(* IEC 61131-3 sources: programs/VI-54/VI-54_20171205/VI-54_20171205/Stations/Screen/LseClass170718/Class/AccessControlCreateAdmin, 1 file *)

(* ---- AccessControlCreateAdmin.st ---- *)
(*!
<Class
	Name               = "AccessControlCreateAdmin"
	Revision           = "1.2"
	RealtimeTask       = "false"
	CyclicTask         = "false"
	BackgroundTask     = "false"
	Sigmatek           = "false"
	OSInterface        = "false"
	HighPriority       = "false"
	Automatic          = "false"
	UpdateMode         = "Prescan"
	SharedCommandTable = "true"
	Objectsize         = "(570,360)"
	Comment            = "class for creating a temporary admin">
	<Channels>
		<Server Name="ClassSvr" Visualized="false" Initialize="false" WriteProtected="true" Retentive="false" Comment="class server"/>
		<Server Name="Create" Visualized="false" Initialize="false" WriteProtected="false" Retentive="false" Comment="write() is the command for creating a Admin user"/>
		<Server Name="Level" Visualized="true" Initialize="true" WriteProtected="false" Retentive="false" Comment="user level default 255 (data channel)"/>
		<Server Name="PassWord" Visualized="true" Initialize="false" WriteProtected="false" Retentive="false" Comment="user password (channel to string object)"/>
		<Server Name="UserName" Visualized="true" Initialize="false" WriteProtected="false" Retentive="false" Comment="user name (channel to string object)"/>
		<Client Name="coAccessControlMain" Required="true" Internal="false" Comment="object channel - Connect to AccessControlMain object"/>
		<Client Name="coSystemLogging" Required="false" Internal="false" Comment="Object channel to SystemLogging (optional)."/>
		<Client Name="StrPassword" Required="true" Internal="true"/>
		<Client Name="StrUsername" Required="true" Internal="true"/>
	</Channels>
	<RevDoku>
		<Owner Company="Sigmatek" Author="BraLis"/>
		<Dokumentation Revision="1.2" Date="2016-05-19" Author="GreJoh" Company="Sigmatek" Description="Client coSystemLogging must not be connected."/>
		<Dokumentation Revision="1.1" Date="2015-09-29" Author="BraLis" Company="Sigmatek" Description="insert the method SystemLogging::LogEventText instead of TRACE-Messages"/>
		<Dokumentation Revision="1.0" Date="2015-09-22" Company="Sigmatek" Description="Creation."/>
	</RevDoku>
	<Network Name="AccessControlCreateAdmin">
		<!-- List of Components in this network -->
		<Components>
			<Object
				Name       = "StrPassword"
				Class      = "String"
				Position   = "(330,510)"
				Visualized = "true">
				<Channels>
					<Server Name="Data"/>
					<Client Name="SingleRealloc" Value="1"/>
				</Channels>
			</Object>
			<Object
				Name       = "StrUsername"
				Class      = "String"
				Position   = "(330,330)"
				Visualized = "true">
				<Channels>
					<Server Name="Data"/>
					<Client Name="SingleRealloc" Value="1"/>
				</Channels>
			</Object>
		</Components>
		<Comments>
		</Comments>
		<!-- List of Connections in this network -->
		<Connections>
			<Connection Source="this.StrUsername" Destination="StrUsername.Data"/>
			<Connection Source="this.StrPassword" Destination="StrPassword.Data"/>
			<Connection Source="this.UserName" Destination="StrUsername.Data" Vertices="(1058,330),(886,420),"/>
			<Connection Source="this.PassWord" Destination="StrPassword.Data" Vertices="(1058,390),(886,600),"/>
		</Connections>
		<!-- Headerfiles -->
		<Options>
		</Options>
	</Network>
</Class>
*)
AccessControlCreateAdmin : CLASS
  //Servers:
	ClassSvr 	: SvrChCmd_DINT;
	Create 	: SvrCh_DINT;
	UserName 	: SvrCh_UDINT;
	PassWord 	: SvrCh_UDINT;
	Level 	: SvrCh_UDINT;
  //Clients:
	coAccessControlMain 	: CltChCmd_AccessControlMain;
	StrUsername 	: CltChCmd_String;
	StrPassword 	: CltChCmd_String;
	coSystemLogging 	: CltChCmd_SystemLogging;
  //Variables:
  //Functions:

	FUNCTION VIRTUAL GLOBAL Create::Write
		VAR_INPUT
			input (EAX) 	: DINT;
		END_VAR
		VAR_OUTPUT
			result (EAX) 	: DINT;
		END_VAR;
  //Tables:
	FUNCTION @STD
		VAR_OUTPUT
			ret_code	: CONFSTATES;
		END_VAR;
	FUNCTION GLOBAL TAB @CT_;
END_CLASS;

#pragma using String
#pragma usingLtd AccessControlMain
#pragma usingLtd SystemLogging

FUNCTION VIRTUAL GLOBAL AccessControlCreateAdmin::Create::Write
	VAR_INPUT
		input (EAX) 	: DINT;
	END_VAR
	VAR_OUTPUT
		result (EAX) 	: DINT;
	END_VAR
  VAR
  	aTmpUsername : ARRAY[0..255] of CHAR;
    aTmpPassword : ARRAY[0..255] of CHAR;
    tmpLenUsername : UDINT;
    tmpLenPassword : UDINT;
  END_VAR

	Create := input;
	result := Create;

  tmpLenUsername := StrUsername.GetLength() + 1;
  tmpLenPassword:= StrPassword.GetLength() + 1;

  if tmpLenUsername > 0 then
    StrUsername.GetDataAt(pData:=#aTmpUsername[0], udSize:=tmpLenUsername, udAt:=0);
    StrPassword.GetDataAt(pData:=#aTmpPassword[0], udSize:=tmpLenPassword, udAt:=0);

    coAccessControlMain.CreateAdmin(pUsername:=#aTmpUsername[0], pPassword:=#aTmpPassword[0], usLevel:=to_usint(Level));
  else
    if IsClientConnected(#coSystemLogging) then
      coSystemLogging.LogEventText("AccessControlCreateAdmin::Create::Write: Kein User angelegt" );
    end_if;

  end_if;

END_FUNCTION
